KUKA KRL program: art_safety.sub

&ACCESS RVP
&COMMENT USER specified PLC program
DEF  art_safety ( )

LOOP
   ARTSafetyDoSPS()
   ARTSysDoStateUpdate()
ENDLOOP

END
